{attribute 'GeneratedUsingTerminal: ELX3252-0000-0016'}
{attribute addProperty BoxType "ELX3252-0000-0016"}
{attribute addProperty Id "AI_Standard_Channel_1AT %I*AI_Standard_Channel_3D09D60D7AI_Standard_Channel_2AT %I*AI_Standard_Channel_3D09D60D7WcStateAT %I*WcState_9091E0EB2InfoDataAT %I*InfoData_94A18F5E2"}
{attribute addProperty CRC "789091926"}
{attribute addProperty Size "18"}
TYPE ELX3252_2F089656 EXTENDS EtcSlaveTerminalBase_947E5A46 :
STRUCT
	{attribute addProperty Name "AI_Standard_Channel_1"}
	AI_Standard_Channel_1 : AI_Standard_Channel_3D09D60D;
	{attribute addProperty Name "AI_Standard_Channel_2"}
	AI_Standard_Channel_2 : AI_Standard_Channel_3D09D60D;
	{attribute addProperty Name "WcState"}
	WcState : WcState_9091E0EB;
	{attribute addProperty Name "InfoData"}
	InfoData : InfoData_94A18F5E;
END_STRUCT
END_TYPE

(* stored: Version 1.2.0.0, ProductVersion 3.1.4024.9
   DUT ELX3252_2F089656: Id {b1c78215-4a48-4299-b9c6-6ec674985c77} *)
